// TIA Portal V16 export
// export: Created 2021-11-12T13:32:47.5570696Z, ExportSetting WithDefaults, DisplayName Totally Integrated Automation Portal, DisplayVersion V16 Update 3, DisplayName TIA Portal Version Control Interface, DisplayVersion V16 Update 2, DisplayName TIA Portal Openness, DisplayVersion V16 Update 3, DisplayName SINAMICS Startdrive Advanced, DisplayVersion V16 Update 5, DisplayName SINAMICS Startdrive G130, G150, S120, S150, SINAMICS MV, S210, DisplayVersion V16 Update 5, DisplayName SINAMICS Startdrive G110M, G120, G120C, G120D, G120P, G115D, DisplayVersion V16 Update 5, DisplayName STEP 7 Professional, DisplayVersion V16 Update 3, DisplayName STEP 7 Safety, DisplayVersion V16, DisplayName WinCC UA Professional, DisplayVersion V16 Update 3
DATA_BLOCK "HMI_PARAM_330"   // DB77
{ S7_Optimized_Access := 'TRUE' }
VERSION : 0.1
// stored: AutoNumber true, DBAccessibleFromOPCUA true, IsOnlyStoredInLoadMemory false, IsRetainMemResEnabled false, IsWriteProtectedInAS false, MemoryReserve 100
   VAR
      xxxxx___BinarySensors___xxxxx : Byte;
      "GL01-BG01" : "UDT_CH_DI_Parameter";   // Reflexní optická závora - Snímání pohybu dílu na dopravníku
      "GL01-BG02" { S7_SetPoint := 'True'} : "UDT_CH_DI_Parameter";   // Reflexní optická závora - Snímání pohybu dílu na dopravníku
      "GL02-BG01" : "UDT_CH_DI_Parameter";   // Reflexní optická závora - Snímání pohybu dílu na dopravníku
      "GL03-BG01" : "UDT_CH_DI_Parameter";   // Reflexní optická závora - Snímání pohybu dílu na dopravníku
      "UC21-FC01_14" : "UDT_CH_DI_Parameter";   // 400V Dopravník ++330 (MK1) OK
      "UC21-FC02_14" : "UDT_CH_DI_Parameter";   // 400V Dopravník ++330 (MK2) OK
      "UC21-FC03_14" : "UDT_CH_DI_Parameter";   // 400V Dopravník ++330 ( MK3) OK
      xxxxx___BinaryOthers___xxxxx : Byte;
      "UH11-SF01_14" : "UDT_CH_DI_Parameter";   // Conveyor Remote
      "UH11-SF01_24" : "UDT_CH_DI_Parameter";   // Conveyor Automat
      "UH11-SF03_14" : "UDT_CH_DI_Parameter";   // Conveyor Start automat
      "UH11-SF04_12" : "UDT_CH_DI_Parameter";   // Conveyor Stop
      "UH11-SF05_14" : "UDT_CH_DI_Parameter";   // Conveyor GL01 Manual Backward
      "UH11-SF05_24" : "UDT_CH_DI_Parameter";   // Conveyor GL01 Manual Forward
      "UH11-SF06_14" : "UDT_CH_DI_Parameter";   // Conveyor GL02 Manual Backward
      "UH11-SF06_24" : "UDT_CH_DI_Parameter";   // Conveyor GL02 Manual Forward
      "UF01-SF02_14" : "UDT_CH_DI_Parameter";   // Conveyor GL03 Manual Backward
      "UF01-SF02_24" : "UDT_CH_DI_Parameter";   // Conveyor GL03 Manual Forward
      "UH11-SF07_14" : "UDT_CH_DI_Parameter";   // Bedna Žádost o výměnu
      "UH11-SF08_14" : "UDT_CH_DI_Parameter";   // Bedna vyměněna
      xxxxx___Drives___xxxxx : Byte;
      "GL01-MA01" : "UDT_Drive1_Parameter";
      "GL02-MA01" : "UDT_Drive1_Parameter";
      "GL03-MA01" : "UDT_Drive1_Parameter";
      "UC21-TA01" : "UDT_SINAMICS_G120_Parameter";
      "UC21-TA02" : "UDT_SINAMICS_G120_Parameter";
      "UC21-TA03" : "UDT_SINAMICS_G120_Parameter";
      xxxxx__Others__xxxxx { S7_SetPoint := 'True'} : Byte;
      CL01 : "UDT_PartCounter_Parameter";   // Bedna na přířezy
      TOF320_GL01_1Tact_PT { S7_SetPoint := 'True'} : Time := T#120s;   // Tof time to stop conv after 320_GL01 stopped
      TOF320_GL01_2Tact_PT : Time := T#120s;   // Tof time to stop conv after 320_GL01 stopped
      TOF330_GL01Tact_PT : Time := T#120s;   // Tof time to stop conv after 330_GL01 stopped
      TOF330_GL02Tact_PT : Time := T#120s;   // Tof time to stop conv after 330_GL02 stopped
      xxxxx__Alarms__xxxxx { S7_SetPoint := 'True'} : Byte;
      CL01_Alarm : "UDT_DI_Mon_Parameter";   // Box full alarm
      CL01_Warn : "UDT_DI_Mon_Parameter";   // Box full warning
      ES : "UDT_DI_Mon_Parameter";   // E-stop
   END_VAR
BEGIN
   "UC21-TA01".RefSpdP2000 := 1500.0;
   "UC21-TA01".RefCurrP2002 := 2.49;
   "UC21-TA01".RefTrqP2003 := 7.29;
   "UC21-TA02".RefSpdP2000 := 1500.0;
   "UC21-TA02".RefCurrP2002 := 2.49;
   "UC21-TA02".RefTrqP2003 := 7.29;
   "UC21-TA03".RefSpdP2000 := 1500.0;
   "UC21-TA03".RefCurrP2002 := 3.6;
   "UC21-TA03".RefTrqP2003 := 14.59;
   CL01_Warn.Func := 16#2;
END_DATA_BLOCK
